(* PLC project PID, Beckhoff Automation GmbH TwinCAT PLC Control 3.5.13.21 *)
(* stored: creationDateTime 2022-05-17T15:59:39.286106, modificationDateTime 2022-05-17T15:59:39.286106 *)

TYPE S_PT1T2_Param :
STRUCT
	K		: REAL;
	T1		: REAL;
	T2		: REAL;
END_STRUCT
END_TYPE
